// TIA Portal V16 export
// export: Created 2025-09-05T07:12:25.751692Z, ExportSetting WithDefaults, DisplayName Totally Integrated Automation Portal, DisplayVersion V16, DisplayName TIA Portal Version Control Interface, DisplayVersion V16, DisplayName TIA Portal Openness, DisplayVersion V16, DisplayName STEP 7 Professional, DisplayVersion V16, DisplayName STEP 7 Safety, DisplayVersion V16, DisplayName WinCC Advanced, DisplayVersion V16
TYPE "UDT WorkStation"
// stored: IsFailsafeCompliant false
   STRUCT
      Status : Struct
         xEntrySensorStatus : Bool;
         xExitSensorStatus : Bool;
         xInProcess : Bool;
         tProcessTime : Time;
         iProcessTimeDone : Int;
      END_STRUCT;
      Command : Struct
         xRequestData : Bool;
      END_STRUCT;
      Fault : Struct
         xSpare : Bool;
      END_STRUCT;
   END_STRUCT;
END_TYPE
